(****************************************************************************************)
(*							Beckhoff Automation Poland									*)
(*							L_TBResetBitOfWord v1.0										*)
(*									29.02.2007											*)
(*				This function resets a single bit in a value of type ”word” to “0”		*)
(*______________________________________________________________________________________*)
FUNCTION L_TBResetBitOfWord : WORD
VAR_INPUT
	wInput: WORD;
	byBitNr: BYTE;
END_VAR
VAR
END_VAR

L_TBResetBitOfWord := wInput;
CASE byBitNr OF
	0:
	L_TBResetBitOfWord.0 := FALSE;
	1:
	L_TBResetBitOfWord.1 := FALSE;
	2:
	L_TBResetBitOfWord.2 := FALSE;
	3:
	L_TBResetBitOfWord.3 := FALSE;
	4:
	L_TBResetBitOfWord.4 := FALSE;
	5:
	L_TBResetBitOfWord.5 := FALSE;
	6:
	L_TBResetBitOfWord.6 := FALSE;
	7:
	L_TBResetBitOfWord.7 := FALSE;
	8:
	L_TBResetBitOfWord.8 := FALSE;
	9:
	L_TBResetBitOfWord.9 := FALSE;
	10:
	L_TBResetBitOfWord.10 := FALSE;
	11:
	L_TBResetBitOfWord.11 := FALSE;
	12:
	L_TBResetBitOfWord.12 := FALSE;
	13:
	L_TBResetBitOfWord.13 := FALSE;
	14:
	L_TBResetBitOfWord.14 := FALSE;
	15:
	L_TBResetBitOfWord.15 := FALSE;
END_CASE

END_FUNCTION

(* stored: Version 1.1.0.1, ProductVersion 3.1.4026.13, FileIdentifier 55e842adcee8395cc5cd2468ec1344588e9a0fbd, FileSignature 7cbd8d8ede3fa32a382570da807035cba9be1db9987bff65998c00a84e98aad0ccae5e344ae12fcece2852c300af697e1580c025a07417929670f07db0834aaa761887240055bb1a21988b6d9abaacdffaa93fc79e2e1b9b8bf6416042bc7bf4eb54792b7788135969aab327886fa62c447cf39986f6f9d39e1293fe55a69e66cd344aea8cca63e47cc8483b32af56640425a7b524cfd268bfe153b29116906820caa8c6250c4a38a82021671d418ca9f3ee0065dadf2f9809feb78a2235a35bde953e659a137dead46ecf27da8283def7df8811d8d902df0a2f67e4c9991385244d68e2d8cecbb6dc96b114a057dbd803d94a799fc90b74a57421820ad618f7
   POU L_TBResetBitOfWord: Id {0da34e6a-ed98-44b3-84ea-856529b75cea}, SpecialFunc None *)
